FUNCTION_BLOCK FB_UpDownSlotS1
VAR_INPUT	
	timeout_up			:LREAL;//MS
	timeout_down		:LREAL;//MS
	extra_down_time		:LREAL;//Ms
	sensor_up			:BOOL;
	sensor_down			:ARRAY[1..16] OF BOOL;

END_VAR
VAR_OUTPUT
	MoveDown_do			:BOOL;
	MoveUp_do			:BOOL;
	Break					:BOOL;//启动提前，停止延后
	anysensor_down		:BOOL;
	state				:INT;
	error_code				:INT;
	error				:BOOL;
END_VAR
VAR
	step				:INT;
	Ton_MoveUp_do		:Tc2_Standard.TON;
	Ton_MoveDown_do		:Tc2_Standard.TON;
	Ton_MoveDown_delay_do :TON;
	ET_Ton_MoveUp_do	:LREAL;
	ET_Ton_MoveDown_do	:LREAL;
	
	i: INT;
	dely_ton_on:Tc2_Standard.TON;//启动时
	dely_ton_off:Tc2_Standard.TON;//关断时
	dely_time:TIME:=T#10MS;
	F_trig_move:Tc2_Standard.F_TRIG;
	en_ton:BOOL;
END_VAR
VAR_IN_OUT
	Initialize			:BOOL;
	MoveDown			:BOOL;
	MoveUp				:BOOL;
	SetOff				:BOOL;
END_VAR

ET_Ton_MoveUp_do:=TIME_TO_LREAL(Ton_MoveUp_do.ET);
ET_Ton_MoveDown_do:=TIME_TO_LREAL(Ton_MoveDown_do.ET);

FOR i:=1 TO 16 DO 
	IF sensor_down[i] THEN 
		anysensor_down:=TRUE;
		EXIT;
	ELSE 
		anysensor_down:=FALSE;
	END_IF
END_FOR

CASE step OF
0://waiting
	IF Initialize THEN 
		step:=5;
	ELSIF MoveDown THEN 
		step:=41;
	ELSIF MoveUp THEN 
		step:=71;
	ELSIF SetOff OR GVL.Reset THEN 
		step:=99;
	END_IF
5://0ff
	MoveDown:=FALSE;
	MoveUp:=FALSE;
	SetOff:=FALSE;
	MoveDown_do:=FALSE;
	MoveUp_do:=FALSE;
	Ton_MoveDown_do(IN:=FALSE , PT:= , Q=> , ET=> );
	Ton_MoveUp_do(IN:=FALSE , PT:= , Q=> , ET=> );
	
	state:=UpDownSlotStateEnum.off;
	error_code:=UpDownSlotErrorEnum.no_error;

	IF Initialize THEN 
		Initialize:=FALSE;		
		step:=10;
	END_IF
10://打开抱闸
	Initialize:=FALSE;
	Break:=TRUE;
	dely_ton_on(IN:=TRUE , PT:=dely_time , Q=> , ET=> );
	IF dely_ton_on.Q THEN 
		dely_ton_on(IN:=FALSE);
		step:=20;
	END_IF

20://初始化，执行上升指令	
	MoveUp_do:=TRUE;	
	MoveUp:=FALSE;
	step:=30;
30://waiting up
	state:=UpDownSlotStateEnum.waiting_up;
	Ton_MoveUp_do(IN:=TRUE , PT:=LREAL_TO_TIME(timeout_up) , Q=> , ET=> );
	IF 	ET_Ton_MoveUp_do>0 AND ET_Ton_MoveUp_do<timeout_up THEN
		IF  sensor_up THEN 			
			MoveUp_do:=FALSE;
			state:=UpDownSlotStateEnum.up;
			Ton_MoveUp_do(IN:=FALSE);
			MoveUp:=FALSE;
			step:=40;				
		END_IF
	ELSIF ET_Ton_MoveUp_do>=timeout_up   THEN 
		IF NOT sensor_up  THEN 
			error_code:=UpDownSlotErrorEnum.timeout_up;
			step:=100;
		END_IF
	END_IF
40://up	
	IF MoveDown  THEN 		
		step:=41;
	END_IF
	(************抱闸***********************)
	dely_ton_off(IN:=TRUE , PT:=dely_time , Q=> , ET=> );
		IF dely_ton_off.Q THEN 
			dely_ton_off(IN:=FALSE);
			Break:=FALSE;
			step:=0;
		END_IF
41://释放抱闸状态		
		IF MoveDown THEN 
			dely_ton_on(IN:=TRUE  , PT:=dely_time , Q=> , ET=> );
			Break:=TRUE;
			IF dely_ton_on.Q THEN 
				dely_ton_on(IN:=FALSE);						
				step:=50;
			END_IF	
		END_IF
50://waiting down
	MoveDown_do:=TRUE;
	MoveDown:=FALSE;
	state:=UpDownSlotStateEnum.waiting_down;
	
	Ton_MoveDown_do(IN:=TRUE , PT:=LREAL_TO_TIME(timeout_down) , Q=> , ET=> );
	IF 	ET_Ton_MoveDown_do>0 AND ET_Ton_MoveDown_do<timeout_down THEN		
		IF  anysensor_down AND NOT sensor_up THEN 
			step:=51;				
		END_IF
	ELSIF ET_Ton_MoveDown_do>=timeout_down  THEN 
		IF NOT  anysensor_down  THEN 
			error_code:=UpDownSlotErrorEnum.timeout_down;
			step:=100;
		END_IF
	END_IF
51://DELAY_DOWN
	Ton_MoveDown_do(IN:=FALSE);
	Ton_MoveDown_delay_do(IN:=TRUE , PT:=LREAL_TO_TIME(extra_down_time) , Q=> , ET=> );
	IF Ton_MoveDown_delay_do.Q THEN 
		Ton_MoveDown_delay_do(IN:=FALSE);
		MoveDown_do:=FALSE;
		state:=UpDownSlotStateEnum.down;
		MoveDown:=FALSE;
		step:=60;	
	END_IF		
	
60://down
	IF MoveUp  THEN 
		step:=20;	
	END_IF
	
	(************抱闸***********************)
	dely_ton_off(IN:=TRUE , PT:=dely_time , Q=> , ET=> );
		IF dely_ton_off.Q THEN 
			dely_ton_off(IN:=FALSE);
			Break:=FALSE;
			step:=0;	
		END_IF	
71://释放 抱闸状态		
		IF MoveUp THEN 
			Break:=TRUE;
			dely_ton_on(IN:=TRUE  , PT:=dely_time , Q=> , ET=> );
			IF dely_ton_on.Q THEN 
				dely_ton_on(IN:=FALSE);							
				step:=20;
			END_IF	
		END_IF
99://setoff
	SetOff:=FALSE;
	error:=FALSE;
	Break:=FALSE;
	MoveDown:=FALSE;
	MoveUp:=FALSE;	
	Initialize:=FALSE;
	MoveDown_do:=FALSE;
	MoveUp_do:=FALSE;
	Ton_MoveDown_do(IN:=FALSE , PT:= , Q=> , ET=> );
	Ton_MoveUp_do(IN:=FALSE , PT:= , Q=> , ET=> );	
	state:=UpDownSlotStateEnum.off;
	error_code:=UpDownSlotErrorEnum.no_error;
	step:=0;
100://error
	error:=TRUE;
	state:=UpDownSlotStateEnum.error;
	MoveUp_do:=FALSE;
	MoveDown_do:=FALSE;
	Break:=FALSE;
	step:=0;	
END_CASE

(************setoff***********************)
IF SetOff OR GVL.Reset THEN 
	step:=99;
END_IF
IF state<>UpDownSlotStateEnum.off AND state<>UpDownSlotStateEnum.error AND  GVL.Emstop_Button THEN 
	error_code:=UpDownSlotErrorEnum.emergency_error;
	step:=100;
END_IF

END_FUNCTION_BLOCK

(* stored: Version 1.1.0.1, ProductVersion 3.1.4024.11
   POU FB_UpDownSlotS1: Id {cf95c4b8-8fb8-4b98-afba-e38ecabe28bf}, SpecialFunc None *)
